// Writes the run as a JUnit XML document - the artifact CI actually consumes.
//
// Implements BOTH reporter faces. I_TestReporter for verdicts and totals,
// I_TestDetailSink for individual checks, because this is the sink that detail
// streaming was designed for: every failed check becomes its own element rather
// than text appended to a growing string.
//
// That is what sidesteps the 255-character ceiling. CONCAT cannot build a longer
// string than that, so a document assembled by concatenation would truncate.
// Assembled as a DOM, no single value ever needs to exceed 255 - the document
// grows by nodes, not by characters.
//
// A DOM rather than streamed text, for one reason above the others: ESCAPING. Test
// labels are author-written and the compared values come from the code under
// test - arbitrary bytes by design. A hand-rolled escape that is subtly wrong
// produces a corrupt document rather than a visible error, and works for a year
// first.
//
// THE WRITE IS ASYNCHRONOUS and driven from CyclicLogic. IsIdle is FALSE until the
// file lands.
//
// ONE RUN, ONE FILE. Nothing is written per suite: a partially written artifact
// read by CI is worse than a missing one, because it looks complete.
FUNCTION_BLOCK TestJUnitReporter IMPLEMENTS I_TestReporter, I_TestDetailSink
VAR
	_Parser : FB_XmlDomParser;

	_RootNode  : SXmlNode;
	_SuiteNode : SXmlNode;
	_CaseNode  : SXmlNode;

	// Node validity is tracked with flags rather than by inspecting SXmlNode. What
	// an unset one contains is not something to rely on.
	_HasDocument  : BOOL;
	_HasSuiteNode : BOOL;
	_HasCaseNode  : BOOL;

	_Path	  : T_MaxString;
	_IsSaving : BOOL;

	_PassedChecks : UDINT;
	_FailedChecks : UDINT;

	// Where a failed write is reported. Never this object's own fan-out - that
	// would call back into here.
	_Reporter : I_TestReporter;

	_FilesWritten	 : UDINT;
	_WriteFailures	 : UDINT;
	_FrameworkErrors : UDINT;
	_LastError		 : HRESULT;
END_VAR

(*
	No cyclic body. CyclicLogic is the cyclic entry point and is called by the
	fan-out, which is called by the suite.
*)

// Where a failed write is reported. Optional but strongly advised.
//
// Without it, the only evidence of a failed write is WriteFailures on this object.
// A sink that cannot write its file and cannot say so is exactly the silence R3
// names.
//
// Deliberately not the fan-out this object is attached to: reporting a write
// failure back through the composite would call this object again.
METHOD AttachErrorSink
VAR_INPUT
	Reporter : I_TestReporter;
END_VAR
_Reporter := Reporter;
END_METHOD

// Start a fresh document. Called on the first result of a run, and again by
// ReRun - a re-run produces a fresh document rather than appending to the last.
METHOD BeginDocument
VAR
	DocumentNode : SXmlNode;
END_VAR
IF _HasDocument THEN
	RETURN;
END_IF

_Parser.NewDocument();

// GetDocumentNode, NOT GetRootNode. The document node is what an element is
// attached to; GetRootNode returns the first ELEMENT, which does not exist yet in
// an empty document. Appending to that one silently does nothing, and the file
// comes out as a bare XML declaration and 23 bytes.
DocumentNode := _Parser.GetDocumentNode();

// The JUnit root. Several suites can sit under it, which is what a sequencer
// produces.
_RootNode	  := _Parser.AppendNode(DocumentNode, 'testsuites');
_HasDocument  := TRUE;
_HasSuiteNode := FALSE;
_HasCaseNode  := FALSE;
END_METHOD

// Open a testsuite element the first time a result arrives for it.
//
// Attributes are filled in at SuiteFinished, when the counts are known - a
// testsuite element carries totals that do not exist while it is running.
METHOD BeginSuite
VAR_INPUT
	SuiteLabel : T_MaxString;
END_VAR
THIS^.BeginDocument();

IF _HasSuiteNode THEN
	RETURN;
END_IF

_SuiteNode	  := _Parser.AppendNode(_RootNode, 'testsuite');
_HasSuiteNode := TRUE;

_Parser.AppendAttribute(_SuiteNode, 'name', SuiteLabel);
END_METHOD

// EVERY failed check gets its own element - not just the first.
//
// This is what the streamed detail was for. The summary keeps only the first
// failure because 80 characters has room for one; the document has room for all of
// them, and each is a separate element rather than a growing string. That
// sidesteps the 255-character ceiling entirely: no single value here can exceed
// it, so nothing has to be truncated to fit.
//
// Expected and Actual go in their own attributes, in full, exactly as they arrived.
METHOD CheckFailed
VAR_INPUT
	StepLabel  : T_MaxString;
	Kind	   : E_FailureKind;
	Expected   : T_MaxString;
	Actual	   : T_MaxString;
	Diagnostic : T_MaxString;
	Message	   : T_MaxString;
END_VAR

VAR
	CheckNode : SXmlNode;
END_VAR
IF NOT _HasCaseNode THEN
	RETURN;
END_IF

_FailedChecks := _FailedChecks + 1;

CheckNode := _Parser.AppendNode(_CaseNode, 'check');

_Parser.AppendAttribute(CheckNode, 'step', StepLabel);
_Parser.AppendAttribute(CheckNode, 'expected', Expected);
_Parser.AppendAttribute(CheckNode, 'actual', Actual);
_Parser.AppendAttribute(CheckNode, 'diagnostic', Diagnostic);
_Parser.AppendAttribute(CheckNode, 'message', Message);
END_METHOD

// Counted, not written. A document listing every satisfied check would be
// enormous and would say nothing a reader wants.
METHOD CheckPassed
VAR_INPUT
	StepLabel : T_MaxString;
	Detail	  : T_MaxString;
END_VAR
_PassedChecks := _PassedChecks + 1;
END_METHOD

// Advances the file write. This is the sink the cyclic method exists for: a DOM
// save is asynchronous and cannot complete in the cycle that asked for it.
//
// SaveDocumentToFile clears the flag it was given when the write finishes, and its
// return value is meaningful on that one call - so the result is captured on the
// transition, not polled for afterwards.
METHOD CyclicLogic
VAR
	Finished : BOOL;
	Written	 : BOOL;
	Error	 : HRESULT;
END_VAR
IF NOT _IsSaving THEN
	RETURN;
END_IF

Written := _Parser.SaveDocumentToFile(sFile := _Path, bExec := _IsSaving,
									  hrErrorCode => Error);

// The method resets _IsSaving when the asynchronous write ends.
Finished := NOT _IsSaving;

IF NOT Finished THEN
	RETURN;
END_IF

// The document has been written, so the next run starts a fresh one. Cleared here
// rather than when the write was requested, so nothing can replace the DOM while
// it is still being read.
_HasDocument := FALSE;

IF Written THEN
	_FilesWritten := _FilesWritten + 1;
	RETURN;
END_IF

// R3: a write that failed is REPORTED, not discarded. The original threw away
// both the FALSE and the HRESULT, which made a bad path indistinguishable from a
// suite that never finished.
_WriteFailures := _WriteFailures + 1;
_LastError	   := Error;

IF _Reporter <> 0 THEN
	_Reporter.FrameworkError('TestJUnitReporter',
		CONCAT('the result document could not be written to ', _Path));
END_IF
END_METHOD

// Size of the document currently in DOM memory, in bytes.
//
// Exposed so a test can prove the document is not EMPTY. Nothing in the PLC can
// read the written file back, and a successful write of an empty document looks
// exactly like a successful write of a full one - which is how a bare 23-byte
// declaration went unnoticed until the file was opened by hand.
PROPERTY DocumentLength : UDINT
GET
DocumentLength := _Parser.GetDocumentLength();
END_GET
END_PROPERTY

// Documents successfully written. One per run.
PROPERTY FilesWritten : UDINT
GET
FilesWritten := _FilesWritten;
END_GET
END_PROPERTY

// Recorded in the document, so a run that could not be trusted says so in the
// artifact rather than only in a log nobody kept.
//
// Not a testcase: it is not a test, and counting it as one would corrupt the
// totals CI reads.
METHOD FrameworkError
VAR_INPUT
	Source	: T_MaxString;
	Message : T_MaxString;
END_VAR

VAR
	ErrorNode : SXmlNode;
END_VAR
THIS^.BeginDocument();

ErrorNode := _Parser.AppendNode(_RootNode, 'framework-error');
_Parser.AppendAttribute(ErrorNode, 'source', Source);
_Parser.AppendAttribute(ErrorNode, 'message', Message);

_FrameworkErrors := _FrameworkErrors + 1;
END_METHOD

PROPERTY FrameworkErrors : UDINT
GET
FrameworkErrors := _FrameworkErrors;
END_GET
END_PROPERTY

// FALSE while the document is being written.
//
// CI must wait for this as well as IsComplete. A run finishing and its file
// reaching disk are different events, and copying between them yields a truncated
// artifact - which reads as a broken pipeline rather than a finished run.
PROPERTY IsIdle : BOOL
GET
IsIdle := NOT _IsSaving;
END_GET
END_PROPERTY

// The failure kind as the string CI groups by. A CASE rather than a lookup table
// because there are six of them and a table would be one more thing to keep in
// step with the enum.
METHOD KindName : T_MaxString
VAR_INPUT
	Kind : E_FailureKind;
END_VAR
CASE Kind OF
E_FailureKind.ValueMismatch:
	KindName := 'ValueMismatch';
E_FailureKind.TypeMismatch:
	KindName := 'TypeMismatch';
E_FailureKind.SizeMismatch:
	KindName := 'SizeMismatch';
E_FailureKind.Timeout:
	KindName := 'Timeout';
E_FailureKind.Environment:
	KindName := 'Environment';
ELSE
	KindName := 'None';
END_CASE
END_METHOD

// The HRESULT from the most recent failed write, or zero.
PROPERTY LastError : HRESULT
GET
LastError := _LastError;
END_GET
END_PROPERTY

// Every suite is done. Requests the write.
//
// The document is NOT written per suite. One run, one file - a partially written
// artifact read by CI is worse than a missing one, because it looks complete.
METHOD RunFinished
VAR_INPUT
	Status	   : I_TestRunStatus;
	TargetInfo : T_MaxString;
END_VAR
IF NOT _HasDocument THEN
	// No document was ever opened, which means RunStarted never arrived - this sink
	// was never part of a run. Writing now would invent an artifact for something
	// that did not happen.
	//
	// An EMPTY run is different and does produce a document, carrying tests="0".
	// That was the opposite of the behaviour before RunStarted existed, and the
	// change is deliberate: a missing file is ambiguous - a configuration problem
	// and a run with no tests look identical - while tests="0" says which. It is the
	// same reasoning as R3, one level up.
	RETURN;
END_IF

IF TargetInfo <> '' THEN
	// Which target produced this. Without it a matrix run yields documents that
	// cannot be told apart.
	_Parser.AppendAttribute(_RootNode, 'target', TargetInfo);
END_IF

IF _Path = '' THEN
	IF _Reporter <> 0 THEN
		_Reporter.FrameworkError('TestJUnitReporter',
			'no result path was set - call SetPath at composition');
	END_IF
	_WriteFailures := _WriteFailures + 1;
	RETURN;
END_IF

// CyclicLogic drives it from here. IsIdle stays FALSE until it lands, and CI must
// wait for that as well as IsComplete: a run finishing and its document reaching
// disk are different events.
//
// _HasDocument stays TRUE until the write COMPLETES. Clearing it here would let a
// late notification call BeginDocument and wipe the DOM out from under the write
// in progress.
_IsSaving := TRUE;
END_METHOD

// Opens the document at the start of the run rather than on the first result to
// arrive.
//
// The lazy version worked and was guesswork: it inferred "a run has begun" from
// something happening. This is the run saying so.
METHOD RunStarted
VAR_INPUT
	Label	   : T_MaxString;
	TargetInfo : T_MaxString;
END_VAR
THIS^.BeginDocument();
END_METHOD

// Absolute path of the result document. REQUIRED - there is no default.
//
// The boot folder is where this belongs on a target. On build 4026 the Windows
// location moved to ProgramData - the 4024 path under C:\TwinCAT is wrong and
// writes nowhere useful:
//
//   C:\ProgramData\Beckhoff\TwinCAT\3.1\Boot\TestResults.xml   Windows, 4026
//   /usr/local/etc/TwinCAT/3.1/Boot/TestResults.xml            TwinCAT/BSD
//
// Which is the reason there is no default: the right answer depends on the build
// and the platform, and a wrong one writes somewhere nobody looks.
//
// Deliberately not defaulted. A default that is wrong for the platform writes
// somewhere nobody looks, and a missing file is indistinguishable from a run that
// never finished - the very confusion R3 exists to remove.
METHOD SetPath
VAR_INPUT
	Path : T_MaxString;
END_VAR
_Path := Path;
END_METHOD

// Fills in the totals a testsuite element carries, now that they exist.
METHOD SuiteFinished
VAR_INPUT
	Status : I_TestRunStatus;
END_VAR

VAR
	// AppendAttribute takes its value as VAR_IN_OUT CONSTANT, which needs something
	// with an address. A literal has one; the result of a call does not, so
	// anything computed goes into a local first.
	TimeText : T_MaxString;
END_VAR
IF Status = 0 THEN
	RETURN;
END_IF

THIS^.BeginSuite(Status.Label);

_Parser.AppendAttributeAsUint(_SuiteNode, 'tests', Status.TestCount);
_Parser.AppendAttributeAsUint(_SuiteNode, 'failures', Status.FailedCount);
_Parser.AppendAttributeAsUint(_SuiteNode, 'errors', Status.ErrorCount);
_Parser.AppendAttributeAsUint(_SuiteNode, 'skipped', Status.SkippedCount);
TimeText := LREAL_TO_FMTSTR(Status.TotalDuration, 6, TRUE);
_Parser.AppendAttribute(_SuiteNode, 'time', TimeText);

// The next suite opens its own element. A sequencer driving several produces
// several, all under one testsuites root.
_HasSuiteNode := FALSE;
END_METHOD

// Closes the testcase element with its verdict.
//
// A testcase with no child element is a pass - that is JUnit's convention, not an
// omission. Failure, error and skipped are each a distinct child, because CI
// counts them separately and so should this.
METHOD TestFinished
VAR_INPUT
	SuiteLabel	  : T_MaxString;
	TestLabel	  : T_MaxString;
	Location	  : T_MaxString;
	Status		  : E_TestStatus;
	Kind		  : E_FailureKind;
	Summary		  : T_MaxString;
	ElapsedTime	  : LREAL;
	ElapsedCycles : UDINT;
	Assertions	  : UDINT;
END_VAR

VAR
	VerdictNode : SXmlNode;
	// AppendAttribute takes its value as VAR_IN_OUT CONSTANT, which needs something
	// with an address. A literal has one; the result of a call does not, so
	// anything computed goes into a local first.
	TimeText : T_MaxString;
	TypeText : T_MaxString;
END_VAR
IF NOT _HasCaseNode THEN
	// No TestStarted arrived - a skipped test never becomes active. Open the
	// element now so the result is not lost.
	THIS^.TestStarted(SuiteLabel := SuiteLabel, TestLabel := TestLabel,
					  Location := Location);
END_IF

IF NOT _HasCaseNode THEN
	RETURN;
END_IF

TimeText := LREAL_TO_FMTSTR(ElapsedTime, 6, TRUE);
_Parser.AppendAttribute(_CaseNode, 'time', TimeText);
_Parser.AppendAttributeAsUint(_CaseNode, 'cycles', ElapsedCycles);
_Parser.AppendAttributeAsUint(_CaseNode, 'assertions', Assertions);

// The split, not just the total. A test reporting 12 assertions of which 3 failed
// is a different situation from one reporting 12 that all passed, and the summary
// only ever names the first failure.
_Parser.AppendAttributeAsUint(_CaseNode, 'checks-passed', _PassedChecks);
_Parser.AppendAttributeAsUint(_CaseNode, 'checks-failed', _FailedChecks);

CASE Status OF

E_TestStatus.Failed:
	// AppendChild, not AppendNode: it sets the element's BODY as well as creating
	// it, and the body is what a CI UI shows when someone clicks a failed test. An
	// attribute-only failure displays the message and nothing else.
	//
	// cdata TRUE so the summary needs no escaping of its own - it may contain
	// compared values, which are arbitrary bytes by design.
	VerdictNode := _Parser.AppendChild(_CaseNode, 'failure', Summary, TRUE);

	// The KIND goes in type, which is what CI groups by. The original hardcoded
	// 'AssertionError' for everything and made the field useless.
	TypeText := THIS^.KindName(Kind);
	_Parser.AppendAttribute(VerdictNode, 'type', TypeText);
	_Parser.AppendAttribute(VerdictNode, 'message', Summary);

E_TestStatus.Errored:
	// error, not failure. The code under test was never shown to be wrong, and CI
	// keeps the two apart.
	VerdictNode := _Parser.AppendChild(_CaseNode, 'error', Summary, TRUE);
	TypeText := THIS^.KindName(Kind);
	_Parser.AppendAttribute(VerdictNode, 'type', TypeText);
	_Parser.AppendAttribute(VerdictNode, 'message', Summary);

E_TestStatus.Skipped:
	VerdictNode := _Parser.AppendNode(_CaseNode, 'skipped');

END_CASE

_HasCaseNode := FALSE;
END_METHOD

// A test became the active one. Opens its testcase element, so the checks that
// follow have somewhere to go.
//
// This is why I_TestDetailSink has a TestStarted at all: checks arrive before the
// test has a verdict, and a document builder needs to be told when to open an
// element.
METHOD TestStarted
VAR_INPUT
	SuiteLabel : T_MaxString;
	TestLabel  : T_MaxString;
	Location   : T_MaxString;
END_VAR
THIS^.BeginSuite(SuiteLabel);

_CaseNode	 := _Parser.AppendNode(_SuiteNode, 'testcase');
_HasCaseNode := TRUE;
_FailedChecks := 0;
_PassedChecks := 0;

_Parser.AppendAttribute(_CaseNode, 'name', TestLabel);

// classname is where to LOOK when a test fails. Empty when the test does not
// implement I_TestLocation, which is the common case and not a problem.
_Parser.AppendAttribute(_CaseNode, 'classname', Location);
END_METHOD

// Writes that failed, or were asked for with no path. Never silent - each also
// raises a framework error through the attached sink.
PROPERTY WriteFailures : UDINT
GET
WriteFailures := _WriteFailures;
END_GET
END_PROPERTY

END_FUNCTION_BLOCK

(* stored: Version 1.1.0.1, ProductVersion 3.1.4026.18
   POU TestJUnitReporter: Id {67d7cb68-f77e-4ef3-b270-2de476967aae}, SpecialFunc None
   Folder I_Cyclic: Id {2978ba85-9993-449c-80e4-f695c82302a8}
   Folder I_TestDetailSink: Id {065b6456-bb9a-4d97-bdaf-8e9f3e59ade0}
   Folder I_TestReporter: Id {c489239b-9062-4415-aab2-6766a502963c}
   Method AttachErrorSink: Id {4ada5902-3f35-4826-87be-529cf9bc644b}
   Method BeginDocument: Id {0481c95f-c709-43b3-b386-4bc0e73ea0eb}
   Method BeginSuite: Id {82c27bad-79c6-4653-bcf1-fc8e84fcd6e2}
   Method CheckFailed: Id {a089e327-2f0b-4707-b8b4-52f6eb3bc456}
   Method CheckPassed: Id {c9f314cb-a2d4-46ad-ae38-7b61739f4fb8}
   Method CyclicLogic: Id {adb25844-751c-4681-8f90-ee1cb28cc05b}
   Property DocumentLength: Id {83242637-d7e6-4347-8ba2-ee9ec4607ad2}
   Get Get: Id {26441a2b-2a7b-4390-9862-1333b20e57a8}
   Property FilesWritten: Id {4c430d8d-8b25-49fa-b3b3-06390d203878}
   Get Get: Id {f8fea8cb-3f14-477c-8137-e60bd9c8e290}
   Method FrameworkError: Id {6d3c600d-5bf4-45bd-810d-8c1750fdd3ab}
   Property FrameworkErrors: Id {083ec242-17b4-4e43-a0fa-c7109032cffb}
   Get Get: Id {889d5f55-1ddc-4707-894c-f9c65cfde0c3}
   Property IsIdle: Id {b05a456a-a1f1-452b-9711-ef9fb1a6f3fc}
   Get Get: Id {815ae01a-f03e-4268-bfe0-1671bbd01840}
   Method KindName: Id {58a0baf5-ff3b-4ba1-aea8-616083e7e4ca}
   Property LastError: Id {17db7c7c-f284-4178-a34a-e7e226937625}
   Get Get: Id {84b230ed-7d3c-4ce4-8f4f-8de5fe51e769}
   Method RunFinished: Id {abfac4f1-0da3-4679-a267-2f55b78a7ed0}
   Method RunStarted: Id {64e605b6-2a78-4463-a824-c30b614dc50d}
   Method SetPath: Id {fab71537-94da-4b88-bbea-217beadb4c71}
   Method SuiteFinished: Id {1117e87e-6805-4fc0-9b24-97e9d619cfe0}
   Method TestFinished: Id {f72b67c9-2673-4510-ba51-ea2187bb5faa}
   Method TestStarted: Id {fe57a787-9946-4656-8228-343d1c6d21f2}
   Property WriteFailures: Id {32043aa4-0716-47b1-ac4a-d5fd13766184}
   Get Get: Id {5094ddbb-e39f-452f-8ed4-c6329a53fba8} *)
